FUNCTION_BLOCK ABSTRACT FB_ActorContinous EXTENDS FB_Actor2Point
VAR_INPUT
	fSetPointAutomatic	: REAL; //unit depending setpoint
END_VAR
VAR_OUTPUT
	fOperatingPoint : REAL; //unit depending operating point
END_VAR
VAR
	{attribute 'OPC.UA.DA' := '1'}
	setSetPoint : ST_SetSetPoint;
	{attribute 'OPC.UA.DA' := '1'}
	setPointState : ST_SetPointState;
	
	//internal variables
	fSetPoint	    : REAL; //actual set setpoint
	aSetPointLimits	: ARRAY[1..2] OF REAL; //control mode and unit depending setpoint limits that are set by abstract method SetSetPointLimits() in a subclass 
END_VAR

METHOD MAIN : BOOL
VAR_INPUT
END_VAR
SelectControlMode();
SetSetPointLimits();
SetPointCheck();
END_METHOD

METHOD PROTECTED SelectControlMode : BOOL
VAR_INPUT
END_VAR
SUPER^.SelectControlMode();

//add changing set point to method
IF control.bManualModeActivated THEN
	fsetPoint := setSetPoint.fSetPointManual;
ELSIF control.bAlgorithmModeActivated AND bAlgorithmPermission THEN
	fsetPoint := setSetPoint.fSetPointAlgorithm;
ELSE
	fsetPoint := fSetPointAutomatic;
END_IF
END_METHOD

METHOD PRIVATE SetPointCheck : BOOL
VAR
END_VAR
fSetPoint := MAX(fSetPoint, aSetPointLimits[1]);
fSetPoint := MIN(fSetPoint, aSetPointLimits[2]);
END_METHOD

METHOD PROTECTED ABSTRACT SetSetPointLimits : BOOL
VAR_INPUT
END_VAR
//set control mode depending setpoint limits -> aSetPointLimits
END_METHOD

END_FUNCTION_BLOCK

(* stored: Version 1.1.0.1, ProductVersion 3.1.4024.10
   POU FB_ActorContinous: Id {c8bff7e9-c02c-4471-8259-14c86f2cd564}, SpecialFunc None
   Method MAIN: Id {10fd2c38-d0f2-4506-83f5-f9de93d73f1f}
   Method SelectControlMode: Id {9487b088-9bc5-4a7e-8bf7-9767eafe3f05}
   Method SetPointCheck: Id {a788f595-bc97-42ed-a5e1-110d1f06de83}
   Method SetSetPointLimits: Id {156a380a-be13-4137-b0ba-36981904d328} *)
